PROGRAM MAIN

P_Observer_Pattern();

END_PROGRAM

(* stored: Version 1.1.0.1, ProductVersion 3.1.4024.11
   POU MAIN: Id {0e642115-0087-4ab8-884c-2001d8a42063}, SpecialFunc None *)
